FUNCTION_BLOCK FB_Motor
VAR_INPUT
END_VAR
VAR_OUTPUT
END_VAR
VAR
	//movingup,
//	moving down
//stopped
// slow bit
	InternalState:E_MotorStates;
	slow:BOOL;
END_VAR

METHOD isSlow : BOOL
VAR_INPUT
END_VAR
isSlow:=slow;
END_METHOD

METHOD IsStopped : BOOL
VAR_INPUT
END_VAR
IsStopped:=FALSE;
IF	InternalState=E_MotorStates.stopped	THEN
	IsStopped:=TRUE;
END_IF
END_METHOD

METHOD MoveDown : BOOL
VAR_INPUT
END_VAR
InternalState:=E_MotorStates.movingdown;
slow:=false;
END_METHOD

METHOD MoveUP : BOOL
VAR_INPUT
END_VAR
InternalState:=E_MotorStates.movingup;
slow:=false;
END_METHOD

METHOD SlowDown : BOOL
VAR_INPUT
END_VAR
slow:=true;
END_METHOD

METHOD Stop : BOOL
VAR_INPUT
END_VAR
slow:=FALSE;
InternalState:=E_MotorStates.stopped;
END_METHOD

END_FUNCTION_BLOCK

(* stored: Version 1.1.0.1, ProductVersion 3.1.4024.11
   POU FB_Motor: Id {8ff14de2-fa53-40ce-8077-ab71ae680e4b}, SpecialFunc None
   Method isSlow: Id {f8e84004-ca07-4d7d-8810-55ac664ca33c}
   Method IsStopped: Id {a514c7b1-b3f2-467f-8eb2-ed079e48023e}
   Method MoveDown: Id {51a3ce90-3c02-452f-891c-e66e6e19f2c5}
   Method MoveUP: Id {01223b80-be72-4c65-92ef-96f3c0a2a308}
   Method SlowDown: Id {6d3edecb-0ee9-4c9c-a05b-66a40cdfccc9}
   Method Stop: Id {0dc6ec37-c855-409f-89e7-bd228e45bf11} *)
